PROGRAM P_3Pack
VAR
	nState: INT;
	
	fbTimerConvs: TON;
	fbTimerPickUP: TON;
	fbTimerGrab: TON;
	fbMyTimer4: TON;
	fbMyTimer5: TON;
	fbMyTimer6: TON;
	fbMyTimer7 : TON;
	fbMyTimer8 : TON;
	fbMyTimer9 : TON;
	F_TRIGLid:F_TRIG;
END_VAR

VAR CONSTANT
	Standby: 	INT:=00;
	Start:		INT:=01;
	atEntry: 	INT:=10;
	Moving: 	INT:=20;
	MovingStopLidClamp: INT:=21;
	MovingStopBase: 	INT:=22;
	PickUP: 	INT:=23;
	PickUP2: 	INT:=24;
	Grab: 		INT:=25;
	Grab2: 		INT:=26;
	Drop: 		INT:=27;
	Moving2: 	INT:=28;
	MovingPack: INT:=29;
	RaiseBase:	INT:=65;
	StoppingAtSens: INT:= 67;
	Stopping: 	INT:=40;
	Resetting: 	INT:=50;
	Clamp:		INT:=60;
	Waiting: 	INT:=30;
	Estop: 		INT:=99;
	
	
END_VAR

// This is our third program  in this program we put the lid together with the base so it can be a box.


F_TRIGLid(CLK:=FIO.bPP_LidDetected);  //trigger for the sense at the lid pack

CASE nState OF
	Standby: 
		nState:=Start;
 
	Start:    
		IF FIO.bInConvSorting=TRUE THEN
			FIO.bPP_ConvBase1:=TRUE;
			FIO.bPP_ConvBase2:=TRUE;
			FIO.bPP_ConvLid:=TRUE;
			fbTimerConvs(IN:=TRUE,PT:=T#1S);
			IF fbTimerConvs.Q THEN
			fbTimerConvs(IN:=FALSE); 
			nState:=MovingStopBase;
		END_IF	
	END_IF
	
	MovingStopBase:
			IF FIO.bPP_BaseDetected=TRUE THEN
				FIO.bPP_ConvBase1:=FALSE;						
				nState:=MovingStopLidClamp;			
			END_IF
	
			
	MovingStopLidClamp:	  // where the clam for lid and base are activated.
		IF F_TRIGLid.Q THEN
			FIO.bPP_LidClamp:=TRUE;
			FIO.bPP_BaseClamp:=TRUE;	
			nState:=PickUP;
		END_IF
		
	PickUP:
		IF FIO.bPP_LidClamp=TRUE AND FIO.bPP_BaseClamp=TRUE THEN
			FIO.bPP_ConvBase2:=FALSE;
			FIO.bInConvSorting:=FALSE;
			FIO.bPP_MoveX:=TRUE;
			fbTimerPickUP(IN:=TRUE,PT:=T#2S);
				IF fbTimerPickUP.Q THEN
					fbTimerPickUP(IN:=FALSE); 
					nState:=Grab;
				END_IF
		END_IF
	
	Grab:
		IF FIO.bPP_MoveX=TRUE THEN
			FIO.bPP_ConvLid:=FALSE;
			FIO.bPP_MoveZ:=TRUE;
			FIO.bPP_Grab:=TRUE;
			fbTimerGrab(IN:=TRUE,PT:=T#2S);
				IF fbTimerGrab.Q THEN
					fbTimerGrab(IN:=FALSE);
					FIO.bPP_LidClamp:=FALSE; 
					nState:=Grab2;
				END_IF
		END_IF

	Grab2:
		IF FIO.bPP_Grab=TRUE THEN
			FIO.bPP_MoveZ:=FALSE;
			fbMyTimer4(IN:=TRUE,PT:=T#2S);
				IF fbMyTimer4.Q THEN
					fbMyTimer4(IN:=FALSE); 
					FIO.bPP_MoveX:=FALSE;
					nState:=Drop;	
				END_IF			
		END_IF	
	
	Drop:
		IF FIO.bPP_MoveX=FALSE THEN
		fbMyTimer5(IN:=TRUE,PT:=T#2S);
			IF fbMyTimer5.Q THEN
				fbMyTimer5(IN:=FALSE); 
				FIO.bPP_MoveZ:=TRUE;
				nState:=Moving2;	
			END_IF	
		END_IF		
	
	Moving2:
		IF FIO.bPP_MovingX=FALSE THEN	
		fbMyTimer6(IN:=TRUE,PT:=T#2S);
			IF fbMyTimer6.Q THEN
				fbMyTimer6(IN:=FALSE);
				FIO.bPP_Grab:=FALSE; 
				nState:=MovingPack;	
			END_IF							
		END_IF
	
	MovingPack:
		IF FIO.bPP_Grab=FALSE THEN
			FIO.bPP_MoveZ:=FALSE;
			FIO.bPP_BaseClamp:=FALSE;
			fbMyTimer7(IN:=TRUE,PT:=T#2S);
			IF fbMyTimer7.Q THEN
				fbMyTimer7(IN:=FALSE);
				nState:=RaiseBase;	
			END_IF	
		END_IF
	
	RaiseBase:
		IF FIO.bPP_MoveZ=FALSE THEN
			FIO.bPP_PosRais_Base:=TRUE;
			FIO.bPP_ConvBase2:=TRUE;
			FIO.bPP_ConvOut:=TRUE;
			fbMyTimer8(IN:=TRUE,PT:=T#2S);
			IF fbMyTimer8.Q THEN
				fbMyTimer8(IN:=FALSE);
				FIO.bPP_PosRais_Base:=FALSE;
				nState:=StoppingAtSens;	
			END_IF	
		END_IF
		
	StoppingAtSens:
		IF FIO.bOutPaSens = TRUE THEN
			FIO.bPP_ConvOut:=FALSE;
			nState:=Waiting;
		END_IF
//----------------------------------------------------------------------------//

	Waiting:
			nState:=Standby;
		
//----------------------------------------------------------------------------//		
		
	ELSE
		nState:=9999;	
END_CASE

END_PROGRAM

(* stored: Version 1.1.0.1, ProductVersion 3.1.4024.3
   POU P_3Pack: Id {fe333432-a923-4835-8a79-97f45134b5af}, SpecialFunc None *)
